Omron CX-Programmer project NewProject (CX-Programmer 9.75)

# PLC NewPLC1: CP1L M

## Global symbols (name address type ; comment)
0.00 BOOL  ; START
0.01 BOOL  ; STOP

## Program NewProgram1 (cyclic task 0)

### Section Section1

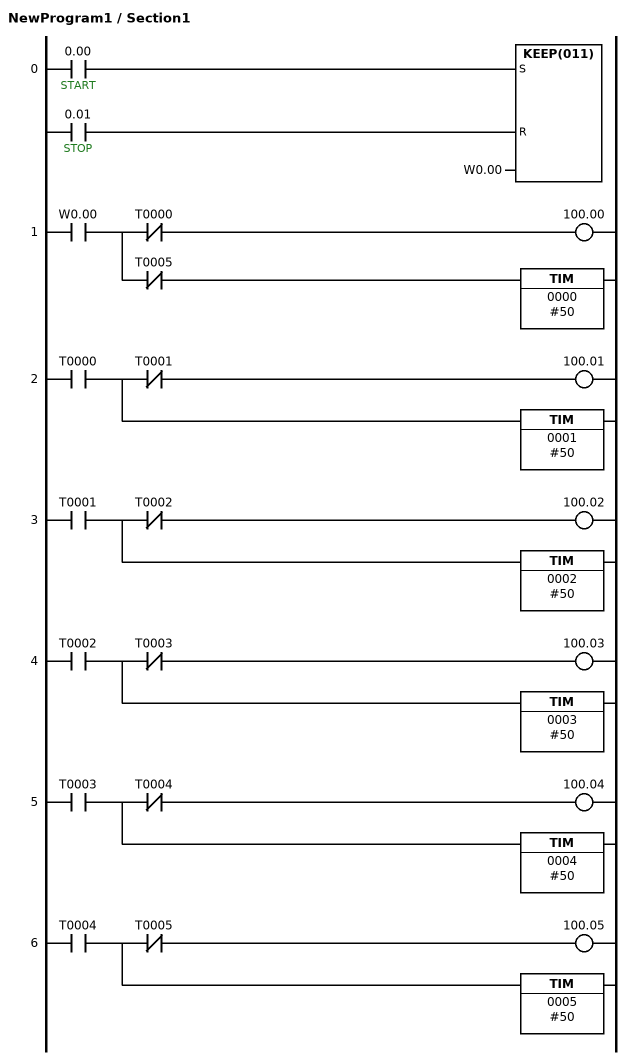
; rung 0
LD 0.00  ; START
LD 0.01  ; STOP
KEEP(011) W0.00
; rung 1
LD W0.00
OUT TR0
ANDNOT T0000
OUT 100.00
LD TR0
ANDNOT T0005
TIM 0000 #50
; rung 2
LD T0000
OUT TR0
ANDNOT T0001
OUT 100.01
LD TR0
TIM 0001 #50
; rung 3
LD T0001
OUT TR0
ANDNOT T0002
OUT 100.02
LD TR0
TIM 0002 #50
; rung 4
LD T0002
OUT TR0
ANDNOT T0003
OUT 100.03
LD TR0
TIM 0003 #50
; rung 5
LD T0003
OUT TR0
ANDNOT T0004
OUT 100.04
LD TR0
TIM 0004 #50
; rung 6
LD T0004
OUT TR0
ANDNOT T0005
OUT 100.05
LD TR0
TIM 0005 #50

### Section END
; rung 0
END(001)